// TIA Portal V19 export
VAR_GLOBAL   // PLC tag table "Sr1000_120"
   unstableReadStatusBits_1_em120 AT %I7019.0 : Bool;
   completionStatusBits_1_em120 AT %I7016.0 : Bool;
   operationInstructionControlBits_1_em120 AT %Q7003.0 : Bool;
   errorStatusBits_1_em120 AT %I7017.0 : Bool;
   busyStatusBits_1_em120 AT %I7015.0 : Bool;
   terminalStatusBits_1_em120 AT %I7018.0 : Bool;
   completionClearControlBits_1_em120 AT %Q7004.0 : Bool;
   handshakeAndGeneralErrorStatusBits_1_em120 AT %I7014.0 : Bool;
   latchAndErrorClearControlBits_1_em120 AT %Q7002.0 : Bool;
   unstableReadStatusByte_1_em120 AT %IB7019 : Byte;
   completionStatusByte_1_em120 AT %IB7016 : Byte;
   operationInstructionControlByte_1_em120 AT %QB7003 : Byte;
   errorStatusByte_1_em120 AT %IB7017 : Byte;
   busyStatusByte_1_em120 AT %IB7015 : Byte;
   terminalStatusByte_1_em120 AT %IB7018 : Byte;
   completionClearControlByte_1_em120 AT %QB7004 : Byte;
   handshakeAndGeneralErrorStatusByte_1_em120 AT %IB7014 : Byte;
   latchAndErrorClearControlByte_1_em120 AT %QB7002 : Byte;
   matchingLevelandTotalEvaluationGradeStatus AT %IB7022 : Byte;
END_VAR
